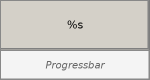
VISUALIZATION UserControlButton  // 150x80
VAR_IN_OUT
	fbButton : FB_Button;
END_VAR
    Button (0,0 150x50), "%s", text variable: fbButton.sButtonName
        tap fbButton.bExecute
        OnMouseDown: execute {  }
    Progressbar (0,50 150x30), variable: fbButton.ExecuteCounter
END_VISUALIZATION

(* stored: Version 1.1.0.1, ProductVersion 3.1.4024.12
   Visu UserControlButton: Id {17cef138-b80a-40d5-ac8b-2cff87a93508} *)
